Omron CX-Programmer project NewProject (CX-Programmer 9.54)

# PLC PLCTry1: CJ2M CPU33
I/O table (CPU CJ2M-CPU33): rack 0 slot 0 CJ1W-ID211; rack 0 slot 1 CJ1W-AD04U-SL; rack 0 slot 2 CJ1W-AD04U-SL; rack 0 slot 11 CJ2M-EIP21

## Global symbols (name address type ; comment)
1.00 BOOL  ; Changes with input temperature

## Program NewProgram1 (cyclic task 0)
Local symbols
CIO2000 BOOL
CIO2001 BOOL
I2000 CHANNEL

### Section Section1

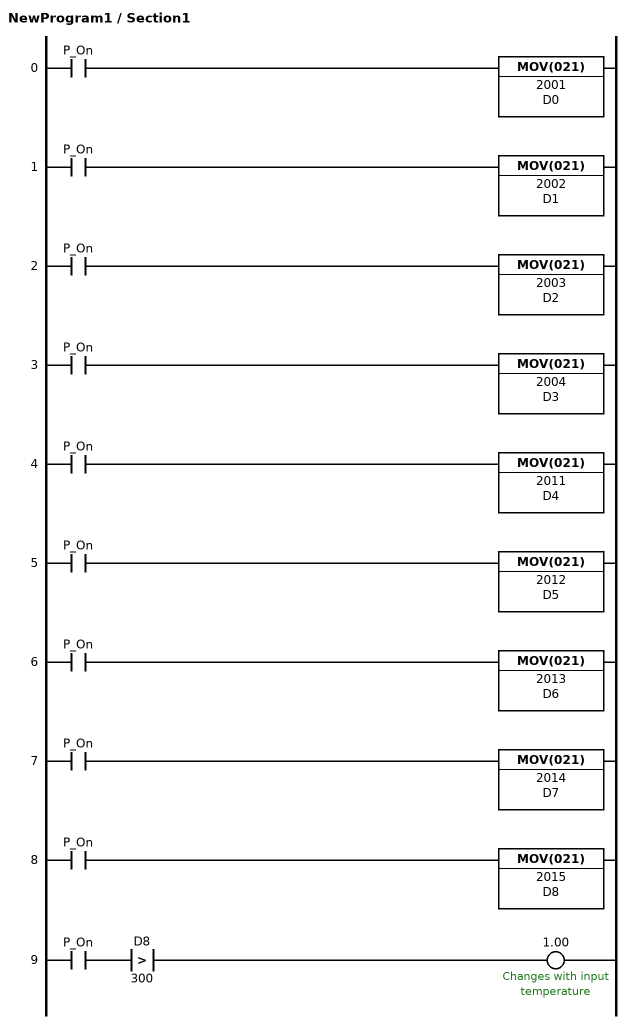
; rung 0
LD P_On
MOV(021) 2001 D0
; rung 1
LD P_On
MOV(021) 2002 D1
; rung 2
LD P_On
MOV(021) 2003 D2
; rung 3
LD P_On
MOV(021) 2004 D3
; rung 4
LD P_On
MOV(021) 2011 D4
; rung 5
LD P_On
MOV(021) 2012 D5
; rung 6
LD P_On
MOV(021) 2013 D6
; rung 7
LD P_On
MOV(021) 2014 D7
; rung 8
LD P_On
MOV(021) 2015 D8
; rung 9
LD P_On
AND>(320) D8 300
OUT 1.00  ; Changes with input temperature

### Section END
; rung 0
END(001)